PROGRAM SafetyMain
VAR
END_VAR

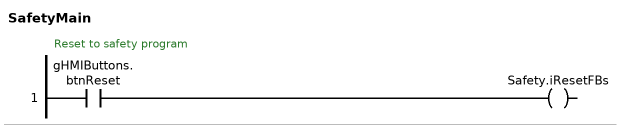
// NETWORK 1
// Reset to safety program
Safety.iResetFBs := gHMIButtons.btnReset;

END_PROGRAM

(* stored: Version 1.1.0.1, ProductVersion 3.1.4024.12
   POU SafetyMain: Id {131003ea-c5f7-4052-9a6a-c5b277ac1841}, SpecialFunc None *)
